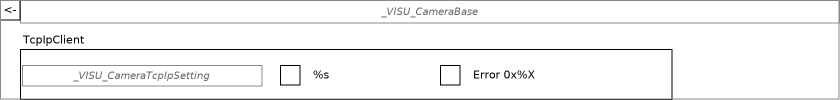
VISUALIZATION _VISU_CameraTcpIp  // 840x100
VAR_IN_OUT
	m_Inst : FB_CameraTcpIp;
END_VAR
    Rectangle (20,49 652x51)
    Frame (20,0 820x23)
        shows _VISU_CameraBase(m_Inst := m_Inst)
    Frame (22,65 240x21)
        shows _VISU_CameraTcpIpSetting(m_Inst := m_Inst)
    RoundedRectangle (0,0 20x20), "<-"
        OnMouseClick: change screen: Previous 
    RoundedRectangle (280,65 20x20), tooltip "Connected", colour toggle: m_Inst._pFbTcpIpClient^.bConnected
    RoundedRectangle (440,65 20x20), tooltip "Connected", colour toggle: m_Inst._pFbTcpIpClient^.bError
    Rectangle (310,65 120x20), "%s", text variable: m_Inst._pFbTcpIpClient^.eStep
    Rectangle (470,65 120x20), "Error 0x%X", text variable: m_Inst._pFbTcpIpClient^.nErrId
    Rectangle (20,30 120x20), "TcpIpClient"
END_VISUALIZATION

(* stored: Version 1.1.0.1, ProductVersion 3.1.4024.3
   Visu _VISU_CameraTcpIp: Id {26e22ab9-1399-4a1f-bd92-35e18c657a94} *)
